TYPE ST_PwrMgmt_HAWino :
STRUCT
	Output	: ST_PwrMgmt_HAWino_In;		// Im Vergleich zur Chargingstation_3 sind hier Input und Output vertauscht!
	Input	: ST_PwrMgmt_HAWino_Out;
END_STRUCT
END_TYPE

(* stored: Version 1.1.0.1, ProductVersion 3.1.4024.11
   DUT ST_PwrMgmt_HAWino: Id {8250481c-da3f-4e88-ad44-e018067d3828} *)
